PROGRAM Vision_Step_ST
VAR
    Always_ON        : BOOL := TRUE;
    Always_OFF       : BOOL := FALSE;

END_VAR

END_PROGRAM

(* stored: Version 1.1.0.1, ProductVersion 3.1.4024.15
   POU Vision_Step_ST: Id {e69f656f-4fbc-4941-803f-6789390cb7a5}, SpecialFunc None *)
